PROGRAM MAIN

END_PROGRAM

(* stored: Version 1.1.0.1, ProductVersion 3.1.4024.4
   POU MAIN: Id {0701205e-8042-4eb2-9ac5-9191561a1695}, SpecialFunc None *)
